PROGRAM MOTION_FB
VAR
	M1: FB_DriveVirtual;
	M1Link: FB_NcAxis;
	bLimitFwdM1 AT %I*: BOOL;
	bLimitBwdM1 AT %I*: BOOL;
	bHomeSensorM1 AT %I*: BOOL;
END_VAR

M1Link(En := TRUE);
M1(En := TRUE,
   bEnable := TRUE,
   bLimitFwd := bLimitFwdM1,
   bLimitBwd := bLimitBwdM1,
   Axis := M1Link.axis);

END_PROGRAM

(* stored: Version 1.1.0.1, ProductVersion 3.1.4020.12
   POU MOTION_FB: Id {069b4de0-b861-4a39-a1ce-08e788017311}, SpecialFunc None *)
